TYPE E_ValveTransitionMode :
(
    Immediate,			// No Condition required, immediate transition
    HoldPrevious_ON,	// OBC Open next valve Before Closing previous
    HoldNext_OFF		// CBO Close previous Before Open next valve
);
END_TYPE

(* stored: Version 1.1.0.1
   DUT E_ValveTransitionMode: Id {f1383028-be09-491a-9f9b-ef4a350deea6} *)
